PROGRAM Digital
VAR
	fbBlinker1: FB_Blinker;
END_VAR

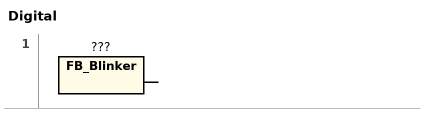
// NETWORK 1
???(); // FB_Blinker

END_PROGRAM

(* stored: Version 1.1.0.1, ProductVersion 3.1.4024.11
   POU Digital: Id {1f8db9e6-24c2-4540-80cf-10cc4334963f}, SpecialFunc None *)
